PROGRAM P_Demo_F_BA_LogMessage2
VAR
    argNLogType                    : DWORD                          := 0; // nLogType
    argSLogCode                    : STRING                         := ''; // sLogCode
    argSLogText                    : T_MaxString                    := ''; // sLogText
    argTArg1                       : T_Arg                         ; // tArg1
    argTArg2                       : T_Arg                         ; // tArg2
END_VAR

// =============================================================================
// Tc3_BA2_Common.F_BA_LogMessage2 演示程序
// =============================================================================
// 场景：`"Setpoint changed from %f to %f"` 两个参数。
//
// 价值：同 LogMessage1，多一参数。
//
// 验证：登录 PLC 后，按例程内变量在线写值；监视输出 / 返回值，结合 §1 功能
//       简述的预期行为对照（详见配套 .md 文档 §7 业务场景）。
//
// 验证步骤：
//   1. 右键 PLC 项目下 POUs 文件夹 → Add → Existing Item → 选本 .TcPOU 文件
//   2. 引用 Tc3_BA2_Common（References → Add library）
//   3. 编译 → 登录 → 运行；按上方『验证』指引在线写值观察
// =============================================================================

fnReturn := F_BA_LogMessage2(
    nLogType                 := argNLogType,
    sLogCode                 := argSLogCode,
    sLogText                 := argSLogText,
    tArg1                    := argTArg1,
    tArg2                    := argTArg2
);

END_PROGRAM

(* stored: Version 1.1.0.1, ProductVersion 3.1.4024.5
   POU P_Demo_F_BA_LogMessage2: Id {20b5c7ea-ba7e-54e5-a6f1-5d95b60c3daf}, SpecialFunc None *)
